// TwinCAT 3 PLC project PLC1
// ProgramVersion: 3.1.4023.0
// libraries:
//   Tc2_Standard, * (Beckhoff Automation GmbH)
//   Tc2_System, * (Beckhoff Automation GmbH)
//   Tc3_Module, * (Beckhoff Automation GmbH)
// project tree:
//   DUTs/ E_State.TcDUT
//   / PlcTask.TcTTO
//   POUs/ FB_StateMachine.TcPOU, MAIN.TcPOU
// real-time tasks:
//   TASK PlcTask: cycle T#10ms, priority 20, ADS port 350

CONFIGURATION PLC1
    RESOURCE PLC ON TwinCAT3
        TASK PlcTask(INTERVAL := T#10ms, PRIORITY := 20);
        PROGRAM MAIN WITH PlcTask : MAIN;
    END_RESOURCE
END_CONFIGURATION

// ---- DUTs/E_State.TcDUT
{attribute 'qualified_only'}
{attribute 'strict'}
TYPE E_State :
(
	Emergency := 0,
	Off := 10,
	Manual := 20,
	Auto := 30,
	CoilClean := 40
);
END_TYPE

// ---- POUs/MAIN.TcPOU
PROGRAM MAIN
VAR
	fbStateMachine : FB_StateMachine;
END_VAR


fbStateMachine();

END_PROGRAM

// ---- POUs/FB_StateMachine.TcPOU
FUNCTION_BLOCK FB_StateMachine
VAR_INPUT
END_VAR
VAR_OUTPUT
END_VAR
VAR
	eState : E_State;
	xManualEnable : BOOL;
	xUnitEnable : BOOL;
	xCoilClean : BOOL;
	xEmergencyFlag : BOOL;
	xCoilCleanFinished : BOOL;
	xFirstCycle: BOOL := TRUE;
END_VAR

IF xFirstCycle THEN 
	eState := E_State.Off;
END_IF
	


CASE eState OF
	
	E_State.Off :
		IF xManualEnable THEN eState := E_State.Manual;
		ELSIF xUnitEnable THEN eState := E_State.Auto;
		END_IF
	
	E_State.Auto :
	 	IF xEmergencyFlag THEN eState := E_State.Emergency;
		ELSIF xManualEnable THEN eState := E_State.Manual;
		ELSIF NOT xUnitEnable THEN eState := E_State.Off;
		END_IF 
	
	E_State.Manual :
		IF NOT xManualEnable THEN eState := E_State.Off;
		ELSIF xCoilClean THEN eState := E_State.CoilClean;					
		END_IF
	
	E_State.CoilClean :
		IF xEmergencyFlag THEN eState := E_State.Emergency;
		ELSIF xCoilCleanFinished THEN eState := E_State.Manual;
									  xCoilClean := FALSE;
									  xCoilCleanFinished := FALSE;								
		END_IF
	
	E_State.Emergency :
		IF NOT xEmergencyFlag THEN eState := E_State.Off;
		END_IF

END_CASE

xFirstCycle := FALSE;

END_FUNCTION_BLOCK
